# EPICS substitutions: OLD/mc11/tpmacApp/pmc/xf23id2-mc11-homing.substitutions
file "home_to_limit_template.pmc"
{

pattern
{ AXIS,   PLC,  SERVO,  TIMER }
{ 1,      8,    701,    5511  }
#{ 2,      9,    702,    5512  }

}
